FUNCTION_BLOCK FB_Module EXTENDS FB_Element IMPLEMENTS I_Module
VAR_INPUT
END_VAR
VAR_OUTPUT
END_VAR
VAR
	fbLogging:					FB_LoggingProvider;
	fbLogger:					FB_Logger<20>;
	{attribute 'OPC.UA.DA' := '1'}
	{attribute 'OPC.UA.DA.Access' := '1'}
	eModeRequest:					E_Mode:= E_Mode.Automatic;				// Requested mod
	{attribute 'OPC.UA.DA' := '1'}
	{attribute 'OPC.UA.DA.Access' := '2'}
	eMode:							E_Mode;				// Current mode
	{attribute 'hide'}
	eModePrevious:					E_Mode;				// Previous mode
	
	fbLevel1:					FB_Level;
	fbLevel2:					FB_Level;
	fbLevel3:					FB_Level;
	fbLevel4:					FB_Level;
END_VAR

// https://peterzerlauth.com/
SUPER^();

fbLevel1();
fbLevel2();
fbLevel3();
fbLevel4();

// Detect mode changes
IF eModeRequest <> E_Mode.Undefined THEN
	IF eMode <> eModeRequest THEN
		eModePrevious:= eMode;
		eMode:= eModeRequest;
		M_OnMode(eMode, eModePrevious);
	END_IF
END_IF
eModeRequest:= E_Mode.Undefined;

METHOD PROTECTED M_Aborting : BOOL (* Return*)
M_Aborting:= 	fbLevel4.M_Request(E_Request.Abort) AND
 				fbLevel3.M_Request(E_Request.Abort) AND
				fbLevel2.M_Request(E_Request.Abort) AND
				fbLevel1.M_Request(E_Request.Abort);
END_METHOD

METHOD PROTECTED M_Completing : BOOL (* Return*)
M_Completing:= 	fbLevel2.M_Request(E_Request.Complete) AND
				fbLevel1.M_Request(E_Request.Complete);
END_METHOD

METHOD PROTECTED M_Holding : BOOL (* Return*)
M_Holding:= fbLevel1.M_Request(E_Request.Hold);
END_METHOD

METHOD PROTECTED M_Idle : BOOL (* Return*)
fbLogging.M_Add(fbLogger);

fbLevel4.P_Event.P_Logger:= fbLogging;
fbLevel3.P_Event.P_Logger:= fbLogging;
fbLevel2.P_Event.P_Logger:= fbLogging;
fbLevel1.P_Event.P_Logger:= fbLogging;

fbLevel4.M_Attach(fbLevel3);
fbLevel4.M_Attach(fbLevel2);
fbLevel4.M_Attach(fbLevel1);

fbLevel3.M_Attach(fbLevel2);
fbLevel3.M_Attach(fbLevel1);

fbLevel2.M_Attach(fbLevel1);

fbEvent.fbObserver.M_Attach(fbLevel1);
END_METHOD

{attribute 'TcRpcEnable':='1'}
METHOD PUBLIC M_Mode : BOOL
VAR_INPUT
	eMode:		E_Mode;
END_VAR
IF THIS^.eMode = eMode THEN
	M_Mode:= TRUE;
ELSE
	eModeRequest:= eMode;	
END_IF
END_METHOD

METHOD PROTECTED M_OnMode
VAR_INPUT
	eMode:							E_Mode;						// Current mode
	eModePrevious:					E_Mode;						// Previous mode	
END_VAR
CASE eMode OF
	E_Mode.Semiauto, E_Mode.Automatic:
		IF eModePrevious = E_Mode.Manual THEN
			fbEvent.M_AddSTRING(TO_STRING(eModePrevious));
			fbEvent.M_AddSTRING(TO_STRING(eMode));
			fbEvent.M_Abort('Module mode changed form %s to %s', 1002);
		END_IF
	E_Mode.Manual:
		;
END_CASE
END_METHOD

METHOD PROTECTED M_Resetting : BOOL (* Return*)
M_Resetting:= 	fbLevel4.M_Request(E_Request.Reset) AND
 				fbLevel3.M_Request(E_Request.Reset) AND
				fbLevel2.M_Request(E_Request.Reset) AND
				fbLevel1.M_Request(E_Request.Reset);
END_METHOD

METHOD PROTECTED M_Starting : BOOL
VAR_INPUT
END_VAR
M_Starting:= 	fbLevel4.M_Request(E_Request.Start) AND_THEN
 				fbLevel3.M_Request(E_Request.Start) AND_THEN
				fbLevel2.M_Request(E_Request.Start) AND_THEN
				fbLevel1.M_Request(E_Request.Start);
END_METHOD

METHOD PROTECTED M_Stopping : BOOL (* Return state complete*)
M_Stopping:= 	fbLevel3.M_Request(E_Request.Stop) AND
				fbLevel2.M_Request(E_Request.Stop) AND
				fbLevel1.M_Request(E_Request.Stop);
END_METHOD

METHOD PROTECTED M_Unholding : BOOL (* Return*)
M_Unholding:= fbLevel1.M_Request(E_Request.Start);
END_METHOD

PROPERTY PUBLIC P_Mode : E_Mode
GET
P_Mode:= eMode;
END_GET
END_PROPERTY

END_FUNCTION_BLOCK

(* stored: Version 1.1.0.1
   POU FB_Module: Id {0d3fc497-598e-0d21-1617-ce19be6391a0}, SpecialFunc None
   Method M_Aborting: Id {1929bb83-c65f-09d2-2a22-b68806b0f4ac}
   Method M_Completing: Id {933fd6f1-4c4e-026e-3128-520b64ab76d5}
   Method M_Holding: Id {ab8a9dd6-7378-063d-2340-22d0380b9c11}
   Method M_Idle: Id {53713e89-9f8a-0ca1-3503-bec2867bc268}
   Method M_Mode: Id {8661b760-0fa5-007a-151c-7fe805544fbb}
   Method M_OnMode: Id {549d817a-659a-0f3e-10ea-6f23f3ce8adf}
   Method M_Resetting: Id {dd412173-49e2-0d05-1622-bbd0077f06b6}
   Method M_Starting: Id {6fe2f334-328e-0cdd-0d07-134e9af3083f}
   Method M_Stopping: Id {36c858d8-accc-01ae-0f5b-a1e3f137f544}
   Method M_Unholding: Id {c789b877-5992-021d-0162-14767b04eb92}
   Property P_Mode: Id {a773e62d-20bd-0c96-369b-0f3305d57073}
   Get Get: Id {0b059178-babf-076f-2ccc-02e13582bfc7} *)
